(* PLC project Beremiz non-standard POUs library, LOLITECH Beremiz 0.0 *)
(* stored: creationDateTime 2008-12-14T16:53:26, modificationDateTime 2009-08-12T15:35:33 *)

FUNCTION_BLOCK GetBoolString
  VAR_INPUT
    VALUE : BOOL;
  END_VAR
  VAR_OUTPUT
    CODE : STRING;
  END_VAR

IF VALUE THEN
  CODE := 'True';
ELSE
  CODE := 'False';
END_IF;
          
END_FUNCTION_BLOCK

FUNCTION_BLOCK TextCtrl
  VAR
    ID : STRING;
  END_VAR
  VAR_INPUT
    back_id : STRING;
    set_text : BOOL;
    text : STRING;
  END_VAR
  VAR
    SVGUI_TEXTCTRL : python_eval;
    setstate_Command : python_eval;
  END_VAR

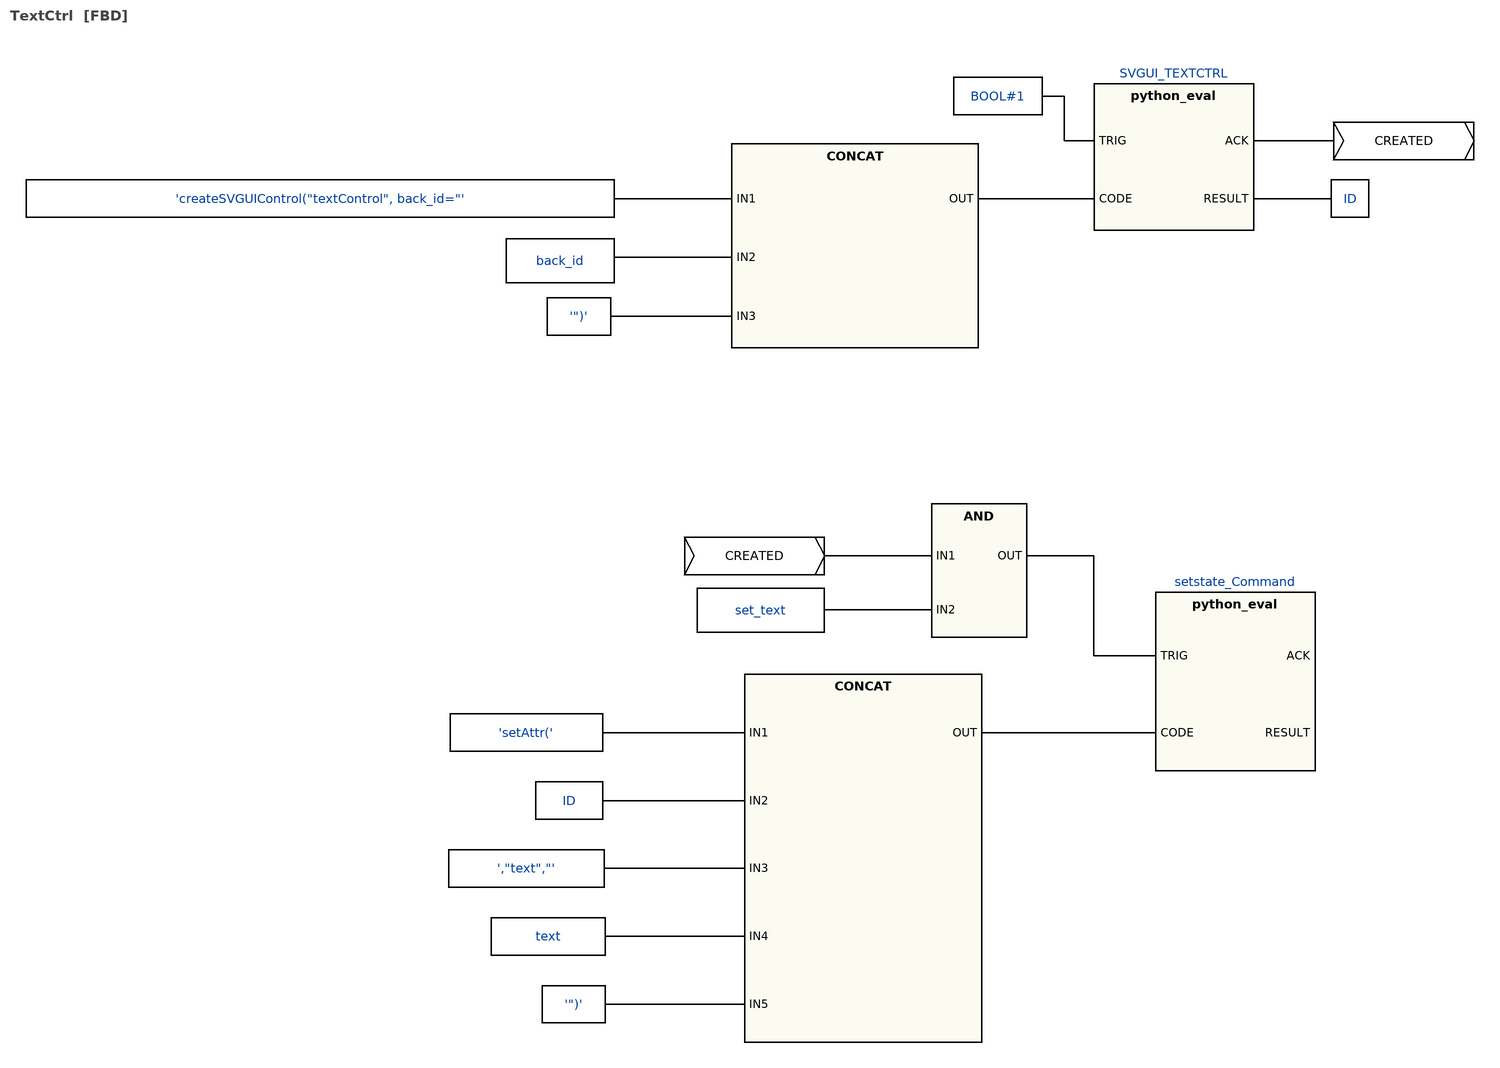
(* FBD diagram, written out as Structured Text *)
SVGUI_TEXTCTRL(TRIG := BOOL#1, CODE := CONCAT('createSVGUIControl("textControl", back_id="', back_id, '")'));
ID := SVGUI_TEXTCTRL.RESULT;
setstate_Command(TRIG := SVGUI_TEXTCTRL.ACK AND set_text, CODE := CONCAT('setAttr(', ID, ',"text","', text, '")'));
END_FUNCTION_BLOCK

FUNCTION_BLOCK Button
  VAR
    ID : STRING;
  END_VAR
  VAR_INPUT
    back_id : STRING;
    sele_id : STRING;
    toggle : BOOL;
    set_state : BOOL;
    state_in : BOOL;
  END_VAR
  VAR_OUTPUT
    state_out : BOOL;
  END_VAR
  VAR
    init_Command : python_eval;
    GetButtonState : GetBoolString;
    setstate_Command : python_eval;
    getstate_Command : python_poll;
    GetButtonToggle : GetBoolString;
  END_VAR

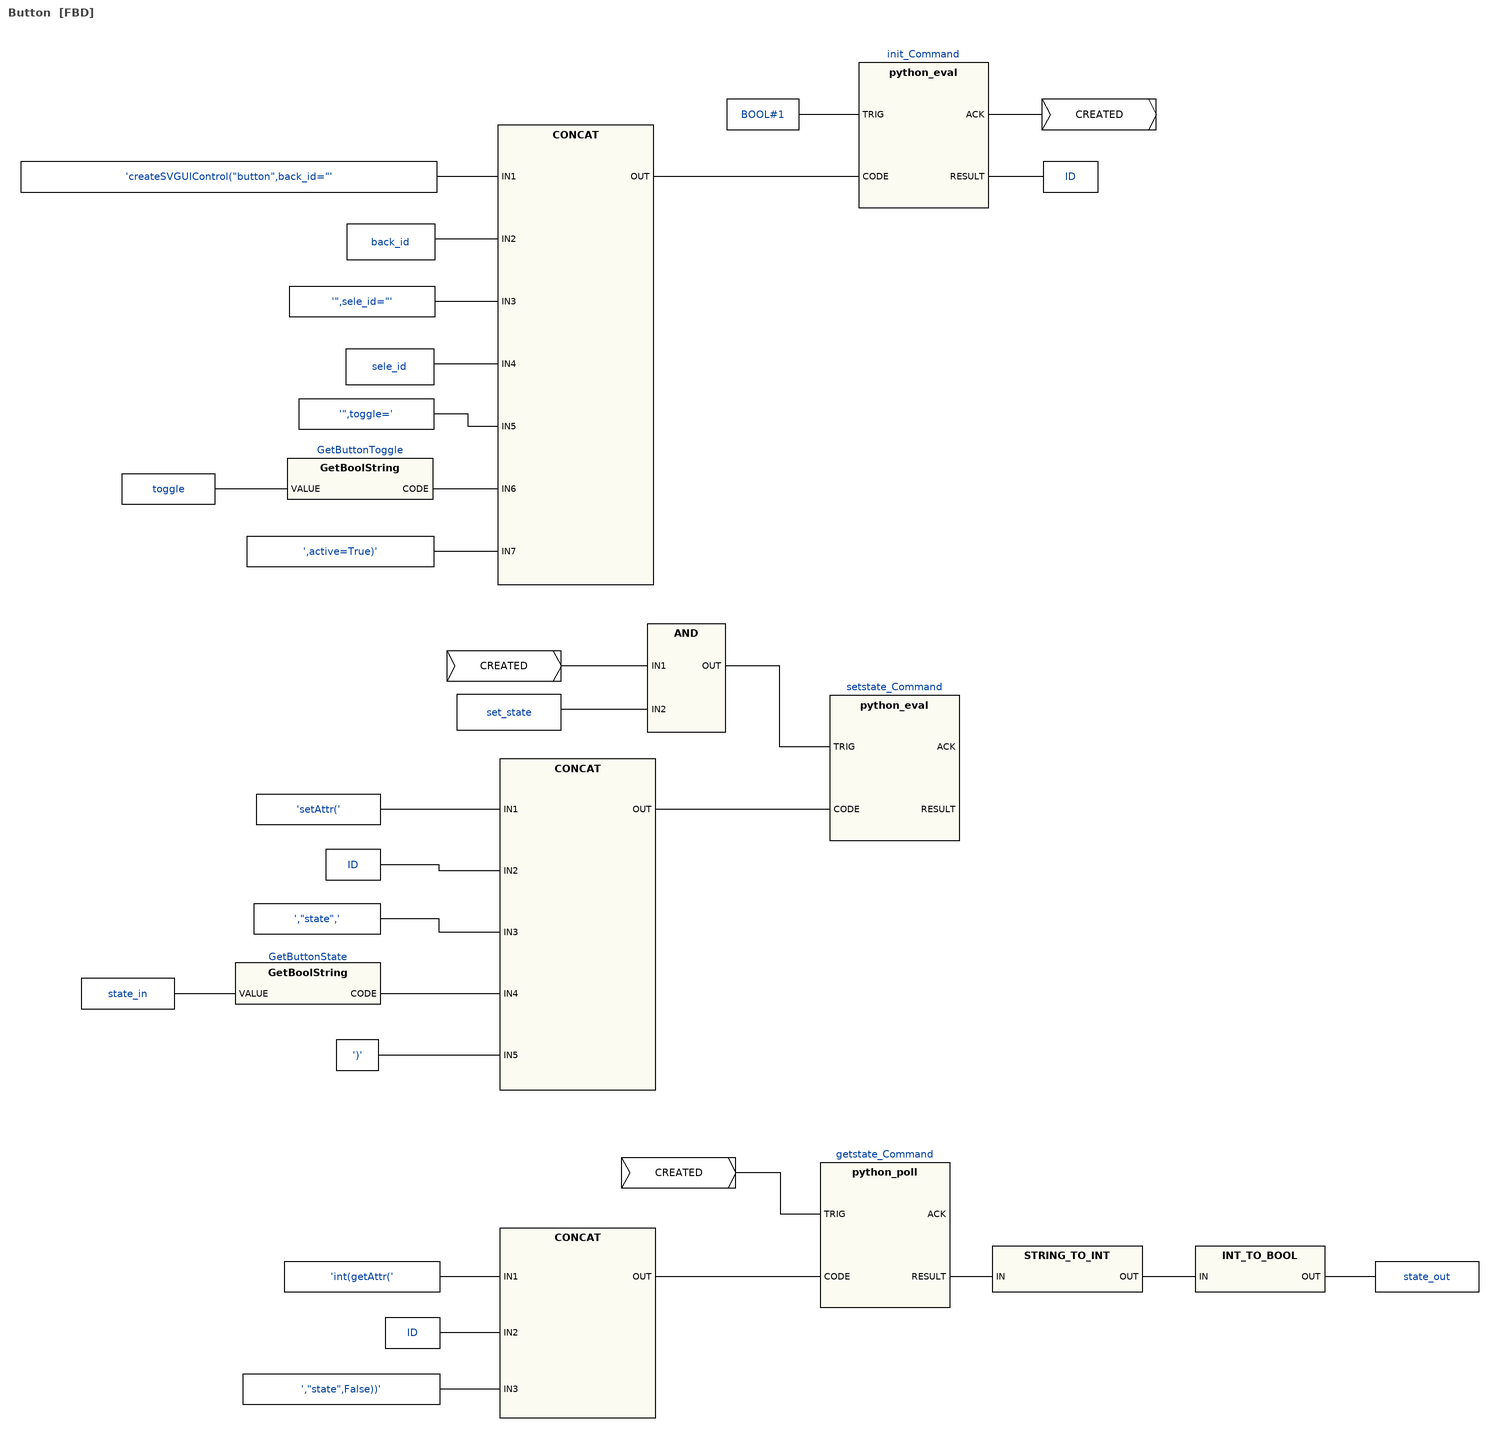
(* FBD diagram, written out as Structured Text *)
GetButtonToggle(VALUE := toggle);
init_Command(TRIG := BOOL#1, CODE := CONCAT('createSVGUIControl("button",back_id="', back_id, '",sele_id="', sele_id, '",toggle=', GetButtonToggle.CODE, ',active=True)'));
ID := init_Command.RESULT;
getstate_Command(TRIG := init_Command.ACK, CODE := CONCAT('int(getAttr(', ID, ',"state",False))'));
state_out := INT_TO_BOOL(STRING_TO_INT(getstate_Command.RESULT));
GetButtonState(VALUE := state_in);
setstate_Command(TRIG := init_Command.ACK AND set_state, CODE := CONCAT('setAttr(', ID, ',"state",', GetButtonState.CODE, ')'));
END_FUNCTION_BLOCK

FUNCTION_BLOCK Led
  VAR
    ID : STRING;
  END_VAR
  VAR_INPUT
    back_id : STRING;
    sele_id : STRING;
    state_in : BOOL;
  END_VAR
  VAR
    init_Command : python_eval;
    setstate_Command : python_poll;
    GetLedState : GetBoolString;
  END_VAR

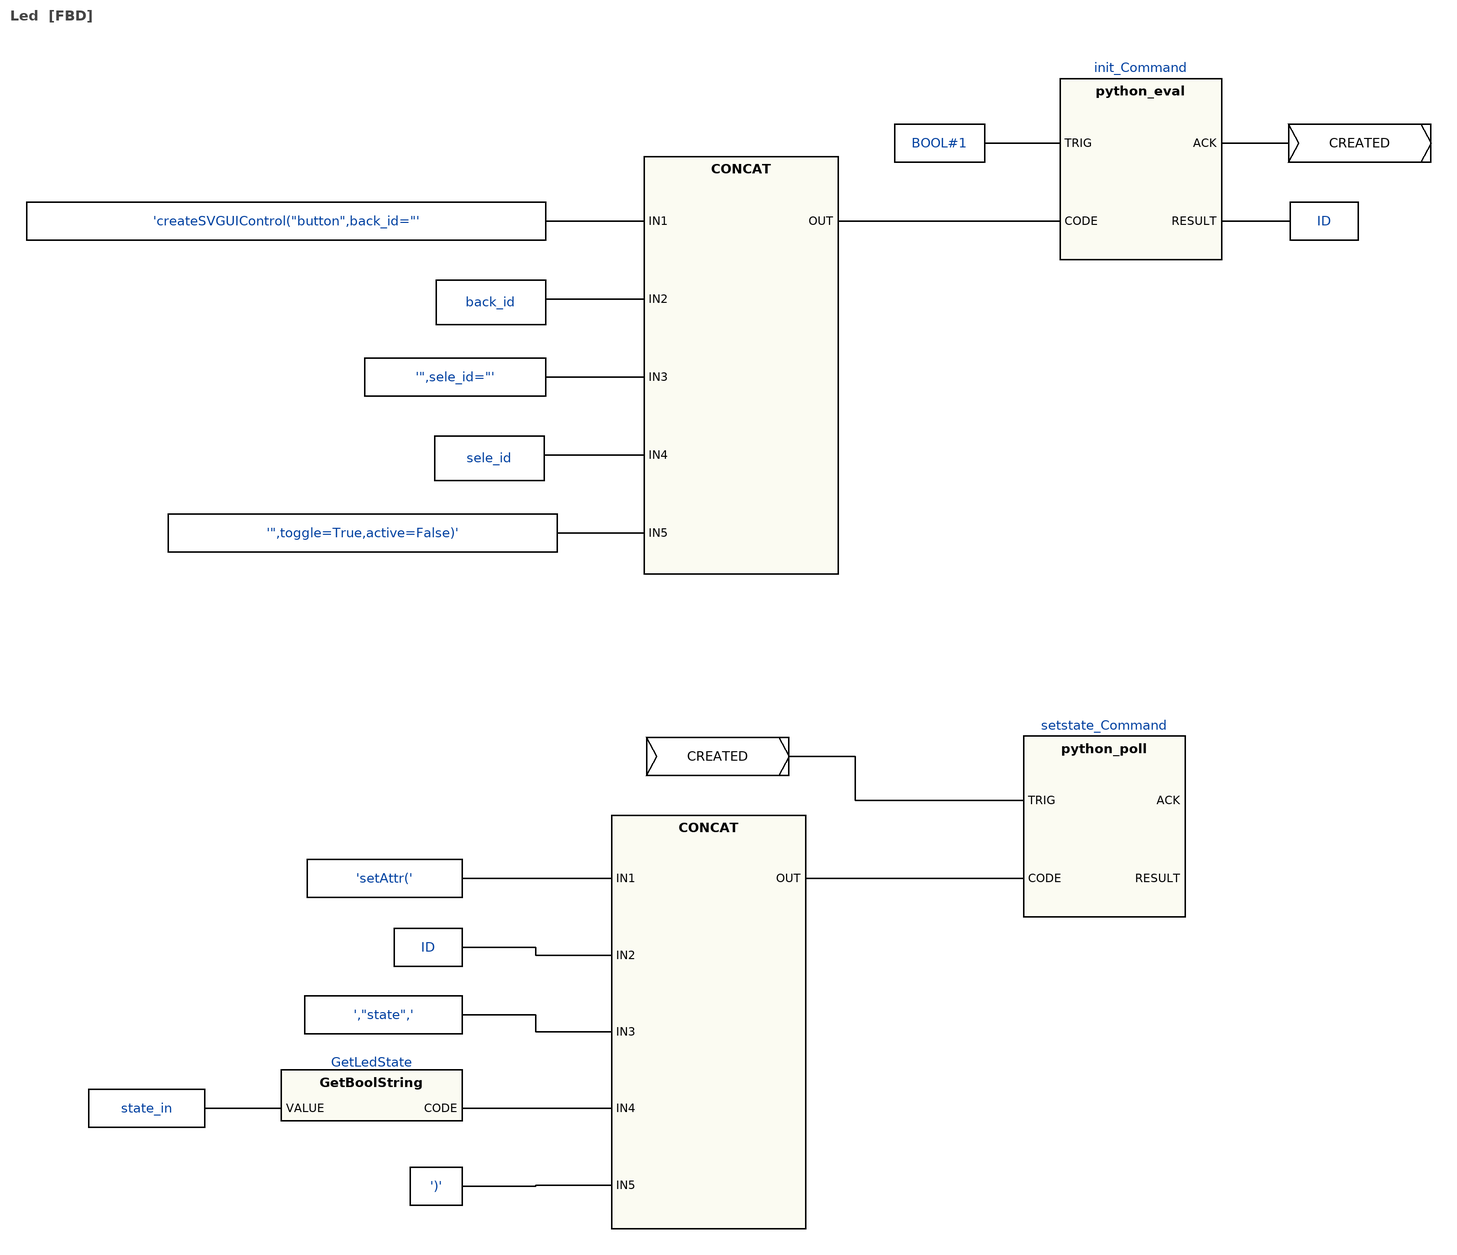
(* FBD diagram, written out as Structured Text *)
init_Command(TRIG := BOOL#1, CODE := CONCAT('createSVGUIControl("button",back_id="', back_id, '",sele_id="', sele_id, '",toggle=True,active=False)'));
ID := init_Command.RESULT;
GetLedState(VALUE := state_in);
setstate_Command(TRIG := init_Command.ACK, CODE := CONCAT('setAttr(', ID, ',"state",', GetLedState.CODE, ')'));
END_FUNCTION_BLOCK
